Omron CX-Programmer project NewProject (CX-Programmer 9.75)

# PLC NewPLC1: CQM1H CPU51

## Global symbols (name address type ; comment)
0.02 BOOL  ; Up/Down Belts Counter
0.10 BOOL  ; machine reset selector]
0.11 BOOL  ; phc before up/down
0.14 BOOL  ; Enter Movable Roller PHC
100.03 BOOL  ; Open/Close Spendels Box 2
100.05 BOOL  ; Open/Close Spendels Box 1
100.09 BOOL  ; Sarin
100.11 BOOL  ; Green Belts Valve
100.13 BOOL  ; Up/Down Valve
101.00 BOOL  ; arm box 2 run
101.01 BOOL  ; arm box 1 run
101.02 BOOL  ; roller under green belts on box 1
101.03 BOOL  ; Fast Movable Roller Green Belts
101.08 BOOL  ; Roller 1 run
101.10 BOOL  ; UP MACHINE
101.11 BOOL  ; DOWN MACHINE
102.00 BOOL  ; roller2 inverter
102.03 BOOL  ; roller under green belts to box 2
102.05 BOOL  ; Green Belts Down
102.07 BOOL  ; work in box 1
102.09 BOOL  ; Green Belts Run
1.01 BOOL  ; Sensor Arm 2 Opend
1.03 BOOL  ; consent from kiln
1.05 BOOL  ; Sensor Box 2 Exiest
1.06 BOOL  ; Fast Up machine
1.08 BOOL  ; Manual Selector
1.11 BOOL  ; start cycle pb
2.05 BOOL  ; Sensor Arm 1 Opend
2.07 BOOL  ; Sensor Box 1 Exiest
50.07 BOOL  ; Machine Up Slow
50.10 BOOL  ; Machine Down Slow
51.01 BOOL  ; NO START PRESS CYCLE
52.06 BOOL  ; Spendels 2 Rotate run
52.07 BOOL  ; Arm valve (open/close)
52.08 BOOL  ; Green belt run manual
52.09 BOOL  ; Roller 1 run manual
53.04 BOOL  ; Roller 2 run manual
56.01 BOOL  ; machine in floor 60
60.00 BOOL  ; up/down valve on
60.05 BOOL  ; up/down valve manual
60.11 BOOL  ; Green Belts Valve up/down manual
70.11 BOOL  ; Machine Stop in fixed roller
CNT020 BOOL  ; time rotate green belt with roller2 speed
DM416 CHANNEL  ; time rotate green belt with roller2 speed
DM417 CHANNEL  ; time start green belts
DM58 CHANNEL  ; Fixed roller floor
DM59 CHANNEL  ; Machine floor
DM804 CHANNEL  ; box floors count
HR0.00 BOOL  ; Machine automatic
HR0.01 BOOL  ; up/down valve  on
HR0.05 BOOL  ; Machine Down Run
HR1.07 BOOL  ; Green Belts Valve
HR6.00 BOOL  ; box 1 working
HR6.01 BOOL  ; box 2 working
HR93.00 BOOL  ; roller1 run
HR98.03 BOOL  ; box 2 arm valve
HR98.07 BOOL  ; box 1 arm valve
HR99.00 BOOL  ; Machine moving
LR0.11 BOOL  ; Start Cycle hmi
LR1.00 BOOL  ; Spendels  1 rotate
LR1.02 BOOL  ; Green Belts Valve up/down
LR1.03 BOOL  ; Green Belts Rotation
LR1.05 BOOL  ; Slow Up machine
LR1.06 BOOL  ; Fast Up Machine
LR1.10 BOOL  ; Slow Down machine
LR1.11 BOOL  ; Fast  Down machine
LR2.00 BOOL  ; Roller 1 Rotation
LR2.01 BOOL  ; Roller 2 Rotation
LR2.03 BOOL  ; choose box 1
LR2.04 BOOL  ; up/down belts run manual
LR2.05 BOOL  ; Spendels 2 Rotate
LR2.06 BOOL  ; Arm Open
LR2.07 BOOL  ; Arm Close
LR2.08 BOOL  ; choose box 2
LR2.09 BOOL  ; Up/down Valve
TIM006 BOOL  ; time up/down on
TIM016 BOOL  ; machine Stop on fixed roller time
TIM019 BOOL  ; machine stop on fixed roller floor
TIM021 BOOL  ; Arms Not Closed Time
TIM060 BOOL  ; time choose box 1
TIM061 BOOL  ; time choose box 2
TIM299 BOOL  ; Start cycle time

## Program NewProgram1 (no task)

### Section Section1

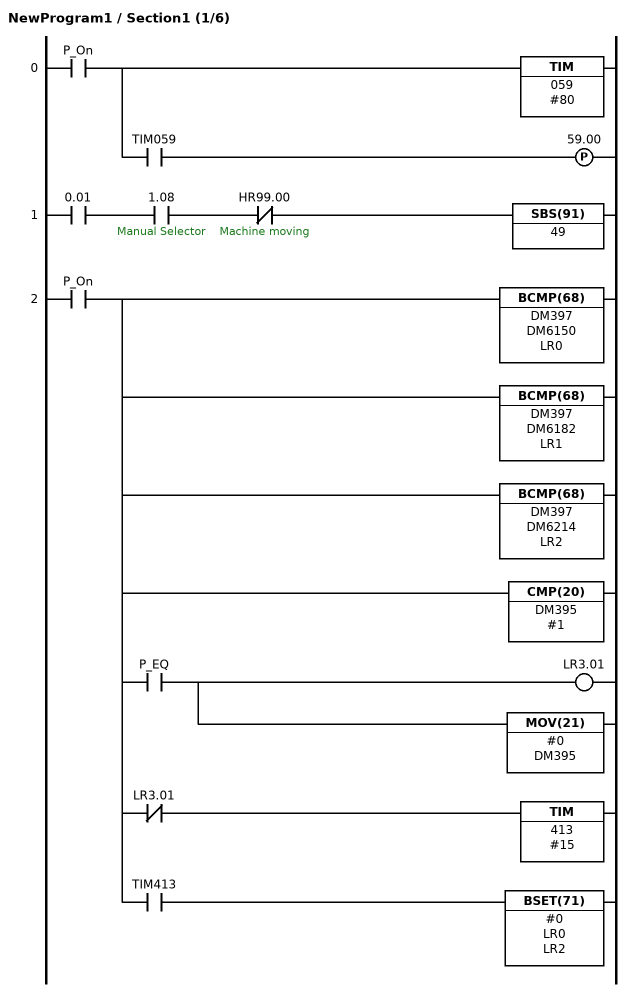
; rung 0
LD P_On
TIM 059 #80
AND TIM059
DIFU(13) 59.00
; rung 1
LD 0.01
AND 1.08  ; Manual Selector
ANDNOT HR99.00  ; Machine moving
SBS(91) 49
; rung 2
LD P_On
OUT TR0
BCMP(68) DM397 DM6150 LR0
BCMP(68) DM397 DM6182 LR1
BCMP(68) DM397 DM6214 LR2
CMP(20) DM395 #1
AND P_EQ
OUT LR3.01
MOV(21) #0 DM395
LD TR0
ANDNOT LR3.01
TIM 413 #15
LD TR0
AND TIM413
BSET(71) #0 LR0 LR2

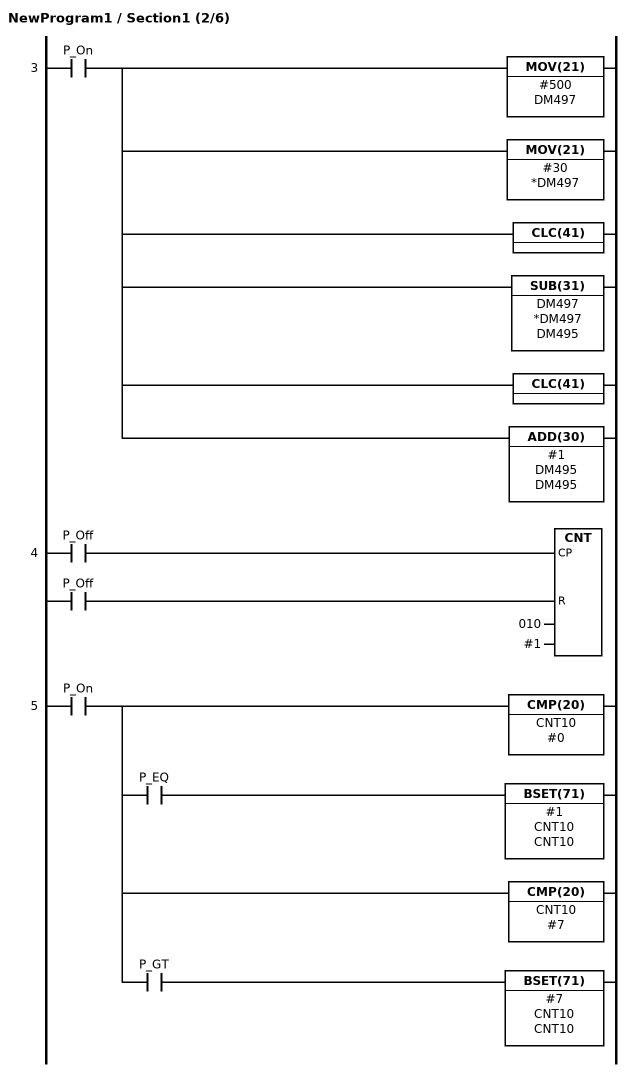
; rung 3
LD P_On
MOV(21) #500 DM497
MOV(21) #30 *DM497
CLC(41)
SUB(31) DM497 *DM497 DM495
CLC(41)
ADD(30) #1 DM495 DM495
; rung 4
LD P_Off
LD P_Off
CNT 010 #1
; rung 5
LD P_On
OUT TR0
CMP(20) CNT10 #0
AND P_EQ
BSET(71) #1 CNT10 CNT10
LD TR0
CMP(20) CNT10 #7
AND P_GT
BSET(71) #7 CNT10 CNT10

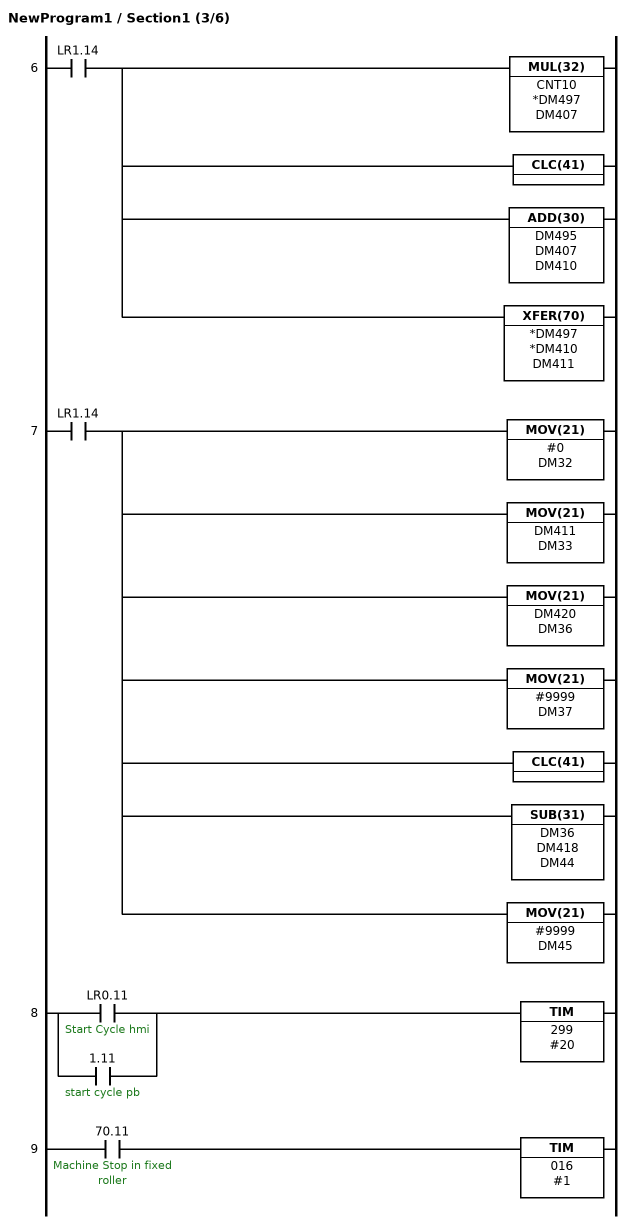
; rung 6
LD LR1.14
MUL(32) CNT10 *DM497 DM407
CLC(41)
ADD(30) DM495 DM407 DM410
XFER(70) *DM497 *DM410 DM411
; rung 7
LD LR1.14
MOV(21) #0 DM32
MOV(21) DM411 DM33
MOV(21) DM420 DM36
MOV(21) #9999 DM37
CLC(41)
SUB(31) DM36 DM418 DM44
MOV(21) #9999 DM45
; rung 8
LD LR0.11  ; Start Cycle hmi
OR 1.11  ; start cycle pb
TIM 299 #20
; rung 9
LD 70.11  ; Machine Stop in fixed roller
TIM 016 #1

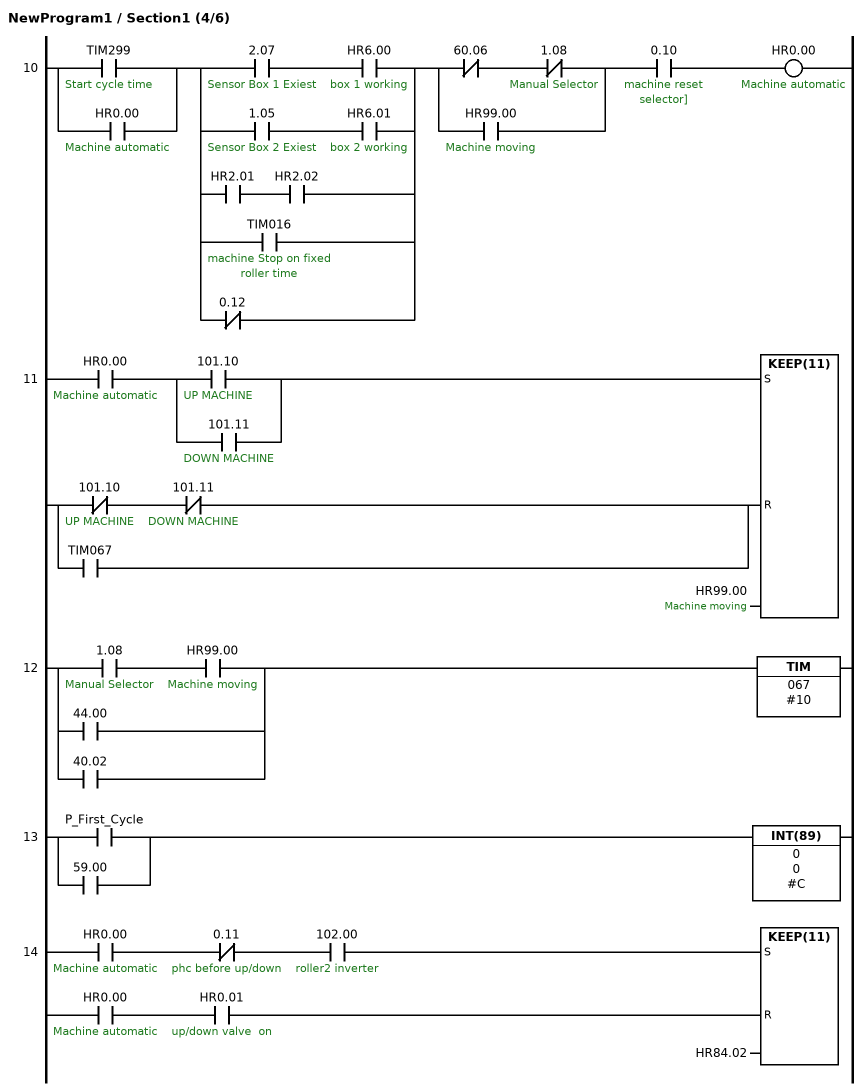
; rung 10
LD TIM299  ; Start cycle time
OR HR0.00  ; Machine automatic
LD 2.07  ; Sensor Box 1 Exiest
AND HR6.00  ; box 1 working
LD 1.05  ; Sensor Box 2 Exiest
AND HR6.01  ; box 2 working
ORLD
LD HR2.01
AND HR2.02
ORLD
OR TIM016  ; machine Stop on fixed roller time
ORNOT 0.12
ANDLD
LDNOT 60.06
ANDNOT 1.08  ; Manual Selector
OR HR99.00  ; Machine moving
ANDLD
AND 0.10  ; machine reset selector]
OUT HR0.00  ; Machine automatic
; rung 11
LD HR0.00  ; Machine automatic
LD 101.10  ; UP MACHINE
OR 101.11  ; DOWN MACHINE
ANDLD
LDNOT 101.10  ; UP MACHINE
ANDNOT 101.11  ; DOWN MACHINE
OR TIM067
KEEP(11) HR99.00  ; Machine moving
; rung 12
LD 1.08  ; Manual Selector
AND HR99.00  ; Machine moving
OR 44.00
OR 40.02
TIM 067 #10
; rung 13
LD P_First_Cycle
OR 59.00
INT(89) 0 0 #C
; rung 14
LD HR0.00  ; Machine automatic
ANDNOT 0.11  ; phc before up/down
AND 102.00  ; roller2 inverter
LD HR0.00  ; Machine automatic
AND HR0.01  ; up/down valve  on
KEEP(11) HR84.02

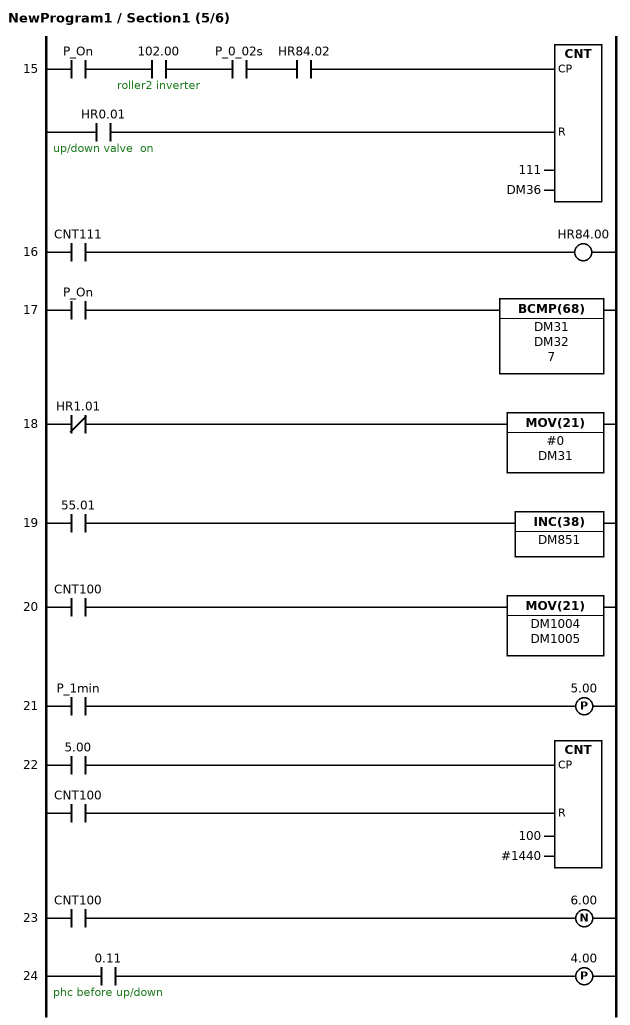
; rung 15
LD P_On
AND 102.00  ; roller2 inverter
AND P_0_02s
AND HR84.02
LD HR0.01  ; up/down valve  on
CNT 111 DM36
; rung 16
LD CNT111
OUT HR84.00
; rung 17
LD P_On
BCMP(68) DM31 DM32 7
; rung 18
LDNOT HR1.01
MOV(21) #0 DM31
; rung 19
LD 55.01
INC(38) DM851
; rung 20
LD CNT100
MOV(21) DM1004 DM1005
; rung 21
LD P_1min
DIFU(13) 5.00
; rung 22
LD 5.00
LD CNT100
CNT 100 #1440
; rung 23
LD CNT100
DIFD(14) 6.00
; rung 24
LD 0.11  ; phc before up/down
DIFU(13) 4.00

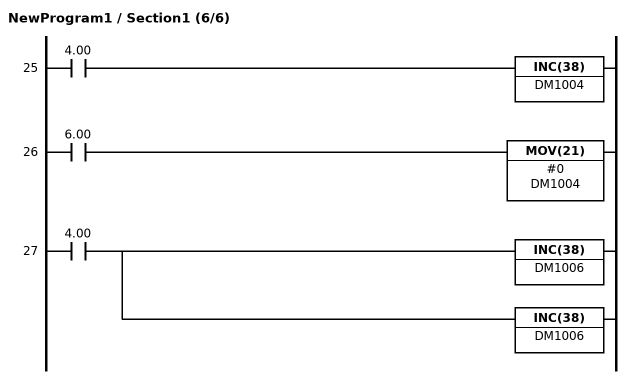
; rung 25
LD 4.00
INC(38) DM1004
; rung 26
LD 6.00
MOV(21) #0 DM1004
; rung 27
LD 4.00
INC(38) DM1006
INC(38) DM1006

### Section Section2

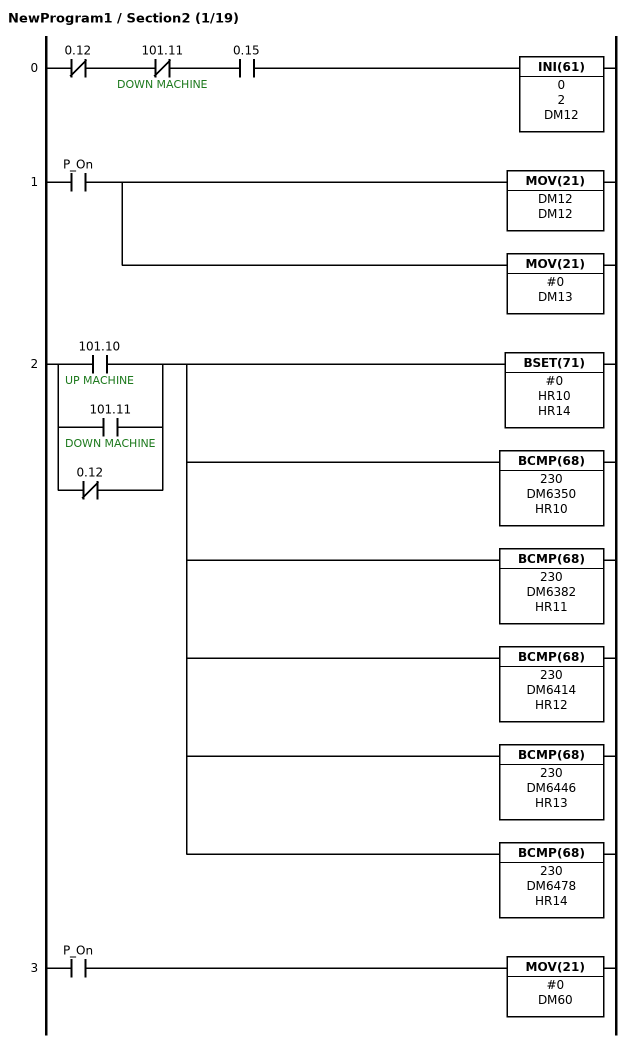
; rung 0
LDNOT 0.12
ANDNOT 101.11  ; DOWN MACHINE
AND 0.15
INI(61) 0 2 DM12
; rung 1
LD P_On
MOV(21) DM12 DM12
MOV(21) #0 DM13
; rung 2
LD 101.10  ; UP MACHINE
OR 101.11  ; DOWN MACHINE
ORNOT 0.12
BSET(71) #0 HR10 HR14
BCMP(68) 230 DM6350 HR10
BCMP(68) 230 DM6382 HR11
BCMP(68) 230 DM6414 HR12
BCMP(68) 230 DM6446 HR13
BCMP(68) 230 DM6478 HR14
; rung 3
LD P_On
MOV(21) #0 DM60

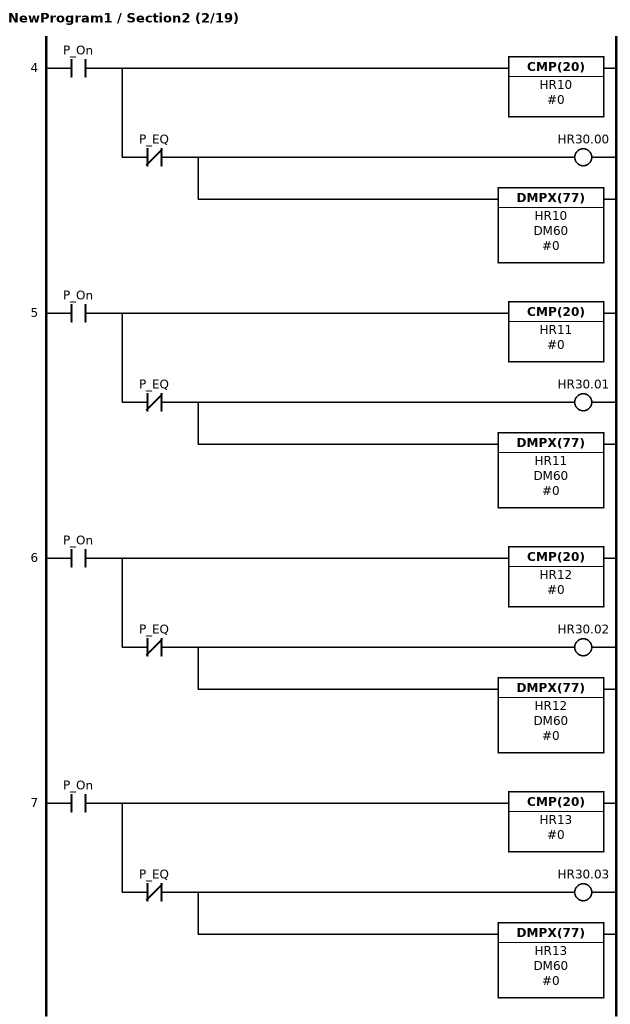
; rung 4
LD P_On
CMP(20) HR10 #0
ANDNOT P_EQ
OUT HR30.00
DMPX(77) HR10 DM60 #0
; rung 5
LD P_On
CMP(20) HR11 #0
ANDNOT P_EQ
OUT HR30.01
DMPX(77) HR11 DM60 #0
; rung 6
LD P_On
CMP(20) HR12 #0
ANDNOT P_EQ
OUT HR30.02
DMPX(77) HR12 DM60 #0
; rung 7
LD P_On
CMP(20) HR13 #0
ANDNOT P_EQ
OUT HR30.03
DMPX(77) HR13 DM60 #0

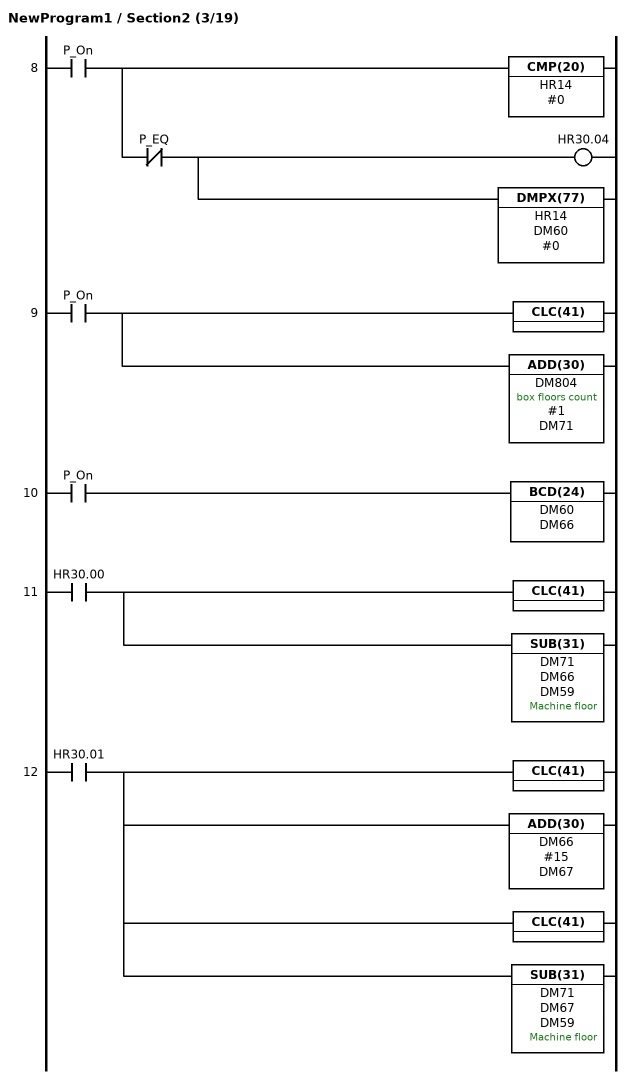
; rung 8
LD P_On
CMP(20) HR14 #0
ANDNOT P_EQ
OUT HR30.04
DMPX(77) HR14 DM60 #0
; rung 9
LD P_On
CLC(41)
ADD(30) DM804 #1 DM71  ; box floors count
; rung 10
LD P_On
BCD(24) DM60 DM66
; rung 11
LD HR30.00
CLC(41)
SUB(31) DM71 DM66 DM59  ; Machine floor
; rung 12
LD HR30.01
CLC(41)
ADD(30) DM66 #15 DM67
CLC(41)
SUB(31) DM71 DM67 DM59  ; Machine floor

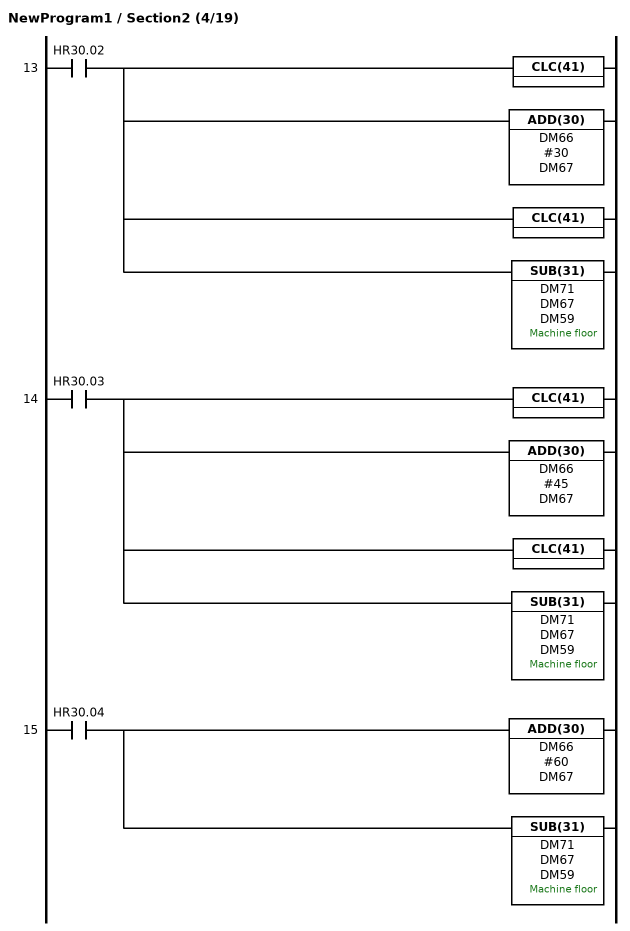
; rung 13
LD HR30.02
CLC(41)
ADD(30) DM66 #30 DM67
CLC(41)
SUB(31) DM71 DM67 DM59  ; Machine floor
; rung 14
LD HR30.03
CLC(41)
ADD(30) DM66 #45 DM67
CLC(41)
SUB(31) DM71 DM67 DM59  ; Machine floor
; rung 15
LD HR30.04
ADD(30) DM66 #60 DM67
SUB(31) DM71 DM67 DM59  ; Machine floor

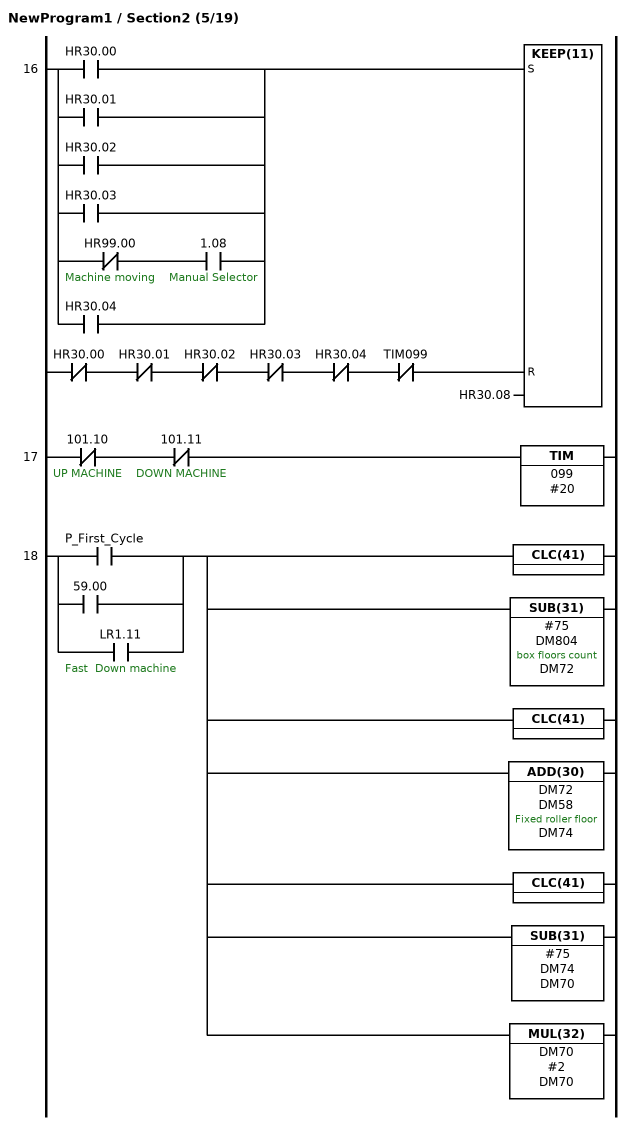
; rung 16
LD HR30.00
OR HR30.01
OR HR30.02
OR HR30.03
LDNOT HR99.00  ; Machine moving
AND 1.08  ; Manual Selector
ORLD
OR HR30.04
LDNOT HR30.00
ANDNOT HR30.01
ANDNOT HR30.02
ANDNOT HR30.03
ANDNOT HR30.04
ANDNOT TIM099
KEEP(11) HR30.08
; rung 17
LDNOT 101.10  ; UP MACHINE
ANDNOT 101.11  ; DOWN MACHINE
TIM 099 #20
; rung 18
LD P_First_Cycle
OR 59.00
OR LR1.11  ; Fast  Down machine
CLC(41)
SUB(31) #75 DM804 DM72  ; box floors count
CLC(41)
ADD(30) DM72 DM58 DM74  ; Fixed roller floor
CLC(41)
SUB(31) #75 DM74 DM70
MUL(32) DM70 #2 DM70

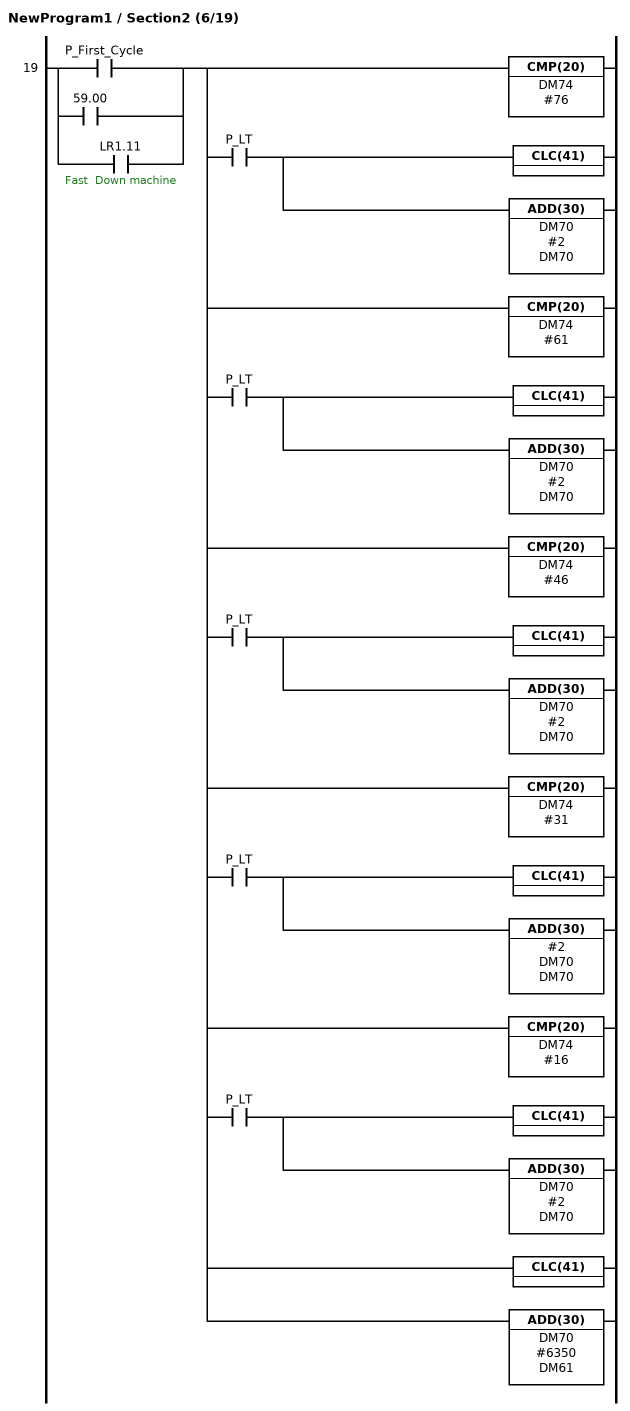
; rung 19
LD P_First_Cycle
OR 59.00
OR LR1.11  ; Fast  Down machine
OUT TR0
CMP(20) DM74 #76
AND P_LT
CLC(41)
ADD(30) DM70 #2 DM70
LD TR0
CMP(20) DM74 #61
AND P_LT
CLC(41)
ADD(30) DM70 #2 DM70
LD TR0
CMP(20) DM74 #46
AND P_LT
CLC(41)
ADD(30) DM70 #2 DM70
LD TR0
CMP(20) DM74 #31
AND P_LT
CLC(41)
ADD(30) #2 DM70 DM70
LD TR0
CMP(20) DM74 #16
AND P_LT
CLC(41)
ADD(30) DM70 #2 DM70
LD TR0
CLC(41)
ADD(30) DM70 #6350 DM61

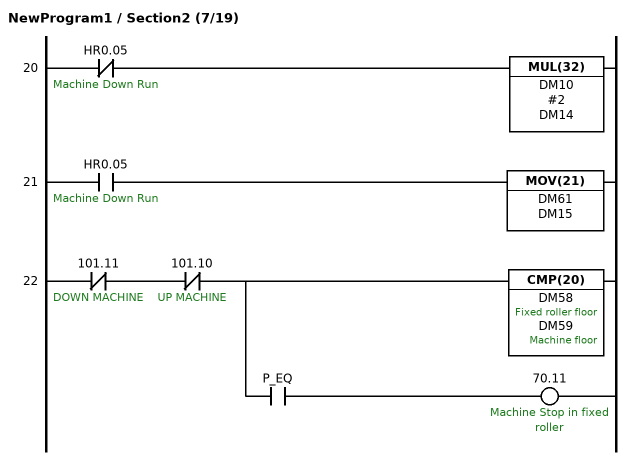
; rung 20
LDNOT HR0.05  ; Machine Down Run
MUL(32) DM10 #2 DM14
; rung 21
LD HR0.05  ; Machine Down Run
MOV(21) DM61 DM15
; rung 22
LDNOT 101.11  ; DOWN MACHINE
ANDNOT 101.10  ; UP MACHINE
CMP(20) DM58 DM59  ; Fixed roller floor, Machine floor
AND P_EQ
OUT 70.11  ; Machine Stop in fixed roller

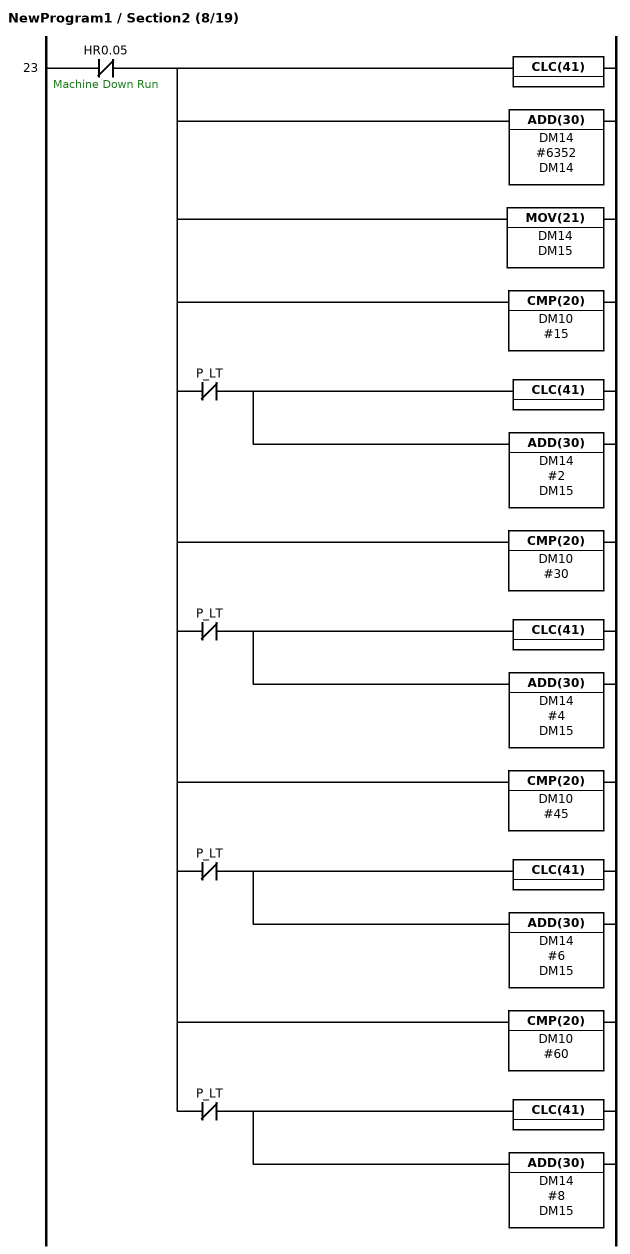
; rung 23
LDNOT HR0.05  ; Machine Down Run
OUT TR0
CLC(41)
ADD(30) DM14 #6352 DM14
MOV(21) DM14 DM15
CMP(20) DM10 #15
ANDNOT P_LT
CLC(41)
ADD(30) DM14 #2 DM15
LD TR0
CMP(20) DM10 #30
ANDNOT P_LT
CLC(41)
ADD(30) DM14 #4 DM15
LD TR0
CMP(20) DM10 #45
ANDNOT P_LT
CLC(41)
ADD(30) DM14 #6 DM15
LD TR0
CMP(20) DM10 #60
ANDNOT P_LT
CLC(41)
ADD(30) DM14 #8 DM15

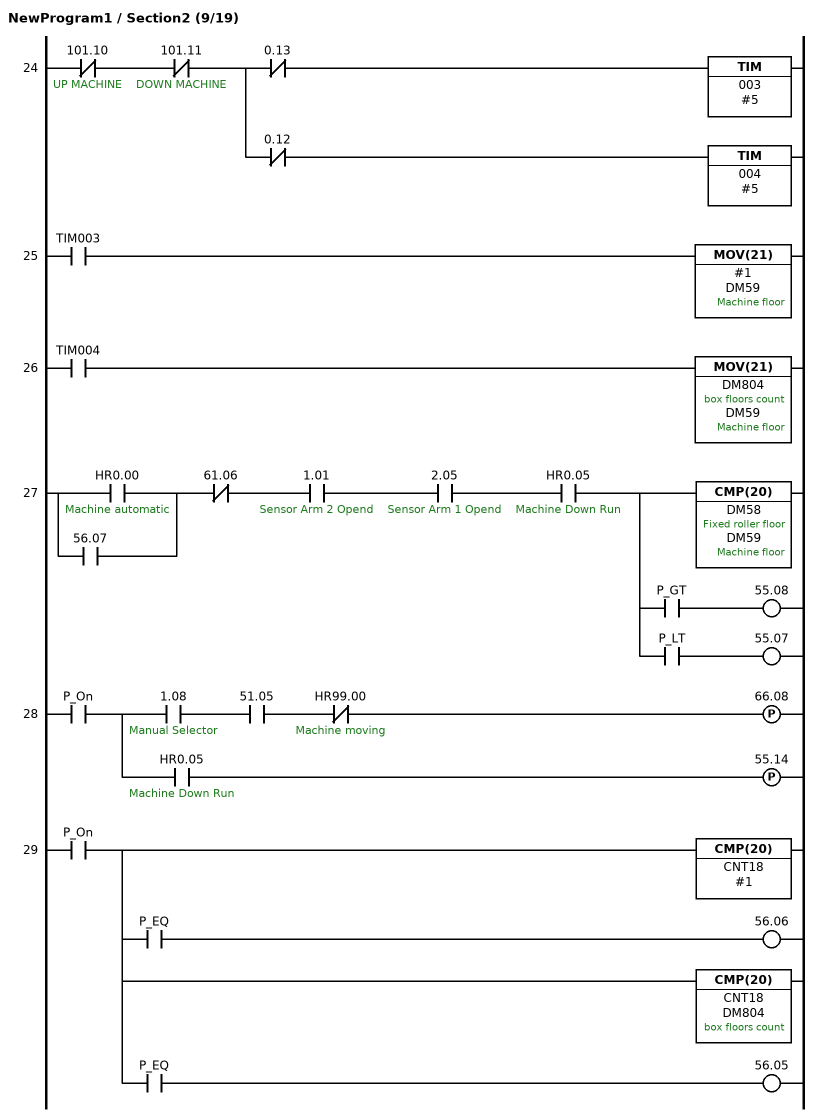
; rung 24
LDNOT 101.10  ; UP MACHINE
ANDNOT 101.11  ; DOWN MACHINE
OUT TR0
ANDNOT 0.13
TIM 003 #5
LD TR0
ANDNOT 0.12
TIM 004 #5
; rung 25
LD TIM003
MOV(21) #1 DM59  ; Machine floor
; rung 26
LD TIM004
MOV(21) DM804 DM59  ; box floors count, Machine floor
; rung 27
LD HR0.00  ; Machine automatic
OR 56.07
ANDNOT 61.06
AND 1.01  ; Sensor Arm 2 Opend
AND 2.05  ; Sensor Arm 1 Opend
AND HR0.05  ; Machine Down Run
OUT TR0
CMP(20) DM58 DM59  ; Fixed roller floor, Machine floor
AND P_GT
OUT 55.08
LD TR0
AND P_LT
OUT 55.07
; rung 28
LD P_On
OUT TR0
AND 1.08  ; Manual Selector
AND 51.05
ANDNOT HR99.00  ; Machine moving
DIFU(13) 66.08
LD TR0
AND HR0.05  ; Machine Down Run
DIFU(13) 55.14
; rung 29
LD P_On
OUT TR0
CMP(20) CNT18 #1
AND P_EQ
OUT 56.06
LD TR0
CMP(20) CNT18 DM804  ; box floors count
AND P_EQ
OUT 56.05

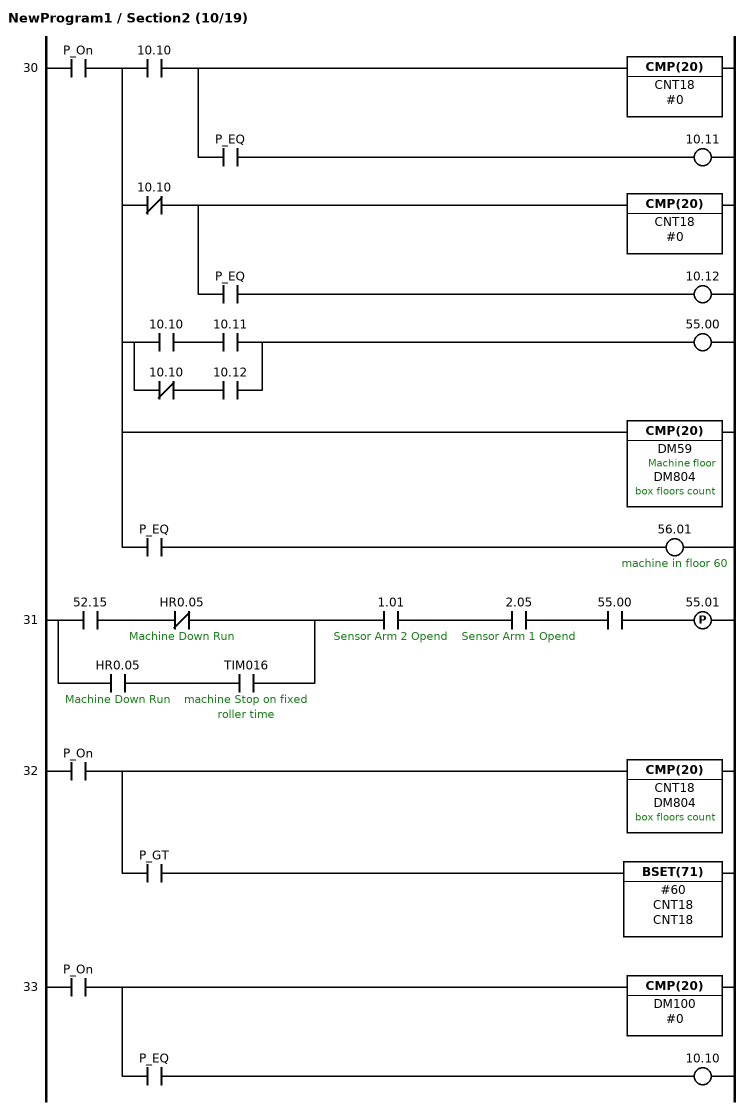
; rung 30
LD P_On
OUT TR0
AND 10.10
CMP(20) CNT18 #0
AND P_EQ
OUT 10.11
LD TR0
ANDNOT 10.10
CMP(20) CNT18 #0
AND P_EQ
OUT 10.12
LD TR0
LD 10.10
AND 10.11
LDNOT 10.10
AND 10.12
ORLD
ANDLD
OUT 55.00
LD TR0
CMP(20) DM59 DM804  ; Machine floor, box floors count
AND P_EQ
OUT 56.01  ; machine in floor 60
; rung 31
LD 52.15
ANDNOT HR0.05  ; Machine Down Run
LD HR0.05  ; Machine Down Run
AND TIM016  ; machine Stop on fixed roller time
ORLD
AND 1.01  ; Sensor Arm 2 Opend
AND 2.05  ; Sensor Arm 1 Opend
AND 55.00
DIFU(13) 55.01
; rung 32
LD P_On
CMP(20) CNT18 DM804  ; box floors count
AND P_GT
BSET(71) #60 CNT18 CNT18
; rung 33
LD P_On
CMP(20) DM100 #0
AND P_EQ
OUT 10.10

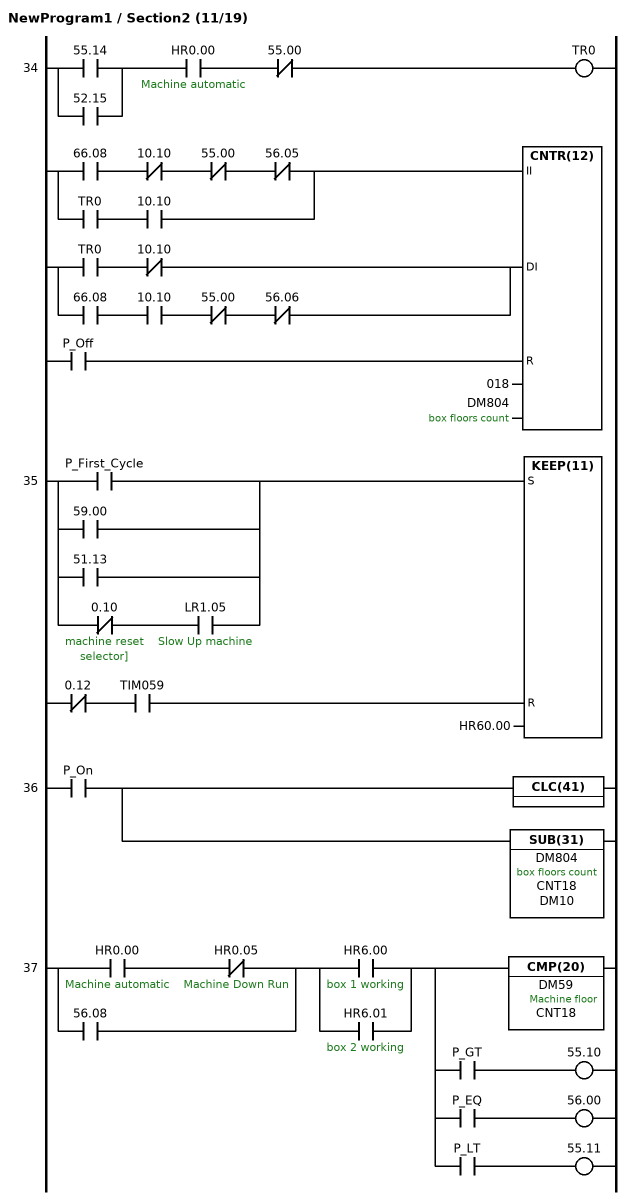
; rung 34
LD 66.08
ANDNOT 10.10
ANDNOT 55.00
ANDNOT 56.05
LD 55.14
OR 52.15
AND HR0.00  ; Machine automatic
ANDNOT 55.00
OUT TR0
AND 10.10
ORLD
LD TR0
ANDNOT 10.10
LD 66.08
AND 10.10
ANDNOT 55.00
ANDNOT 56.06
ORLD
LD P_Off
CNTR(12) 018 DM804  ; box floors count
; rung 35
LD P_First_Cycle
OR 59.00
OR 51.13
LDNOT 0.10  ; machine reset selector]
AND LR1.05  ; Slow Up machine
ORLD
LDNOT 0.12
AND TIM059
KEEP(11) HR60.00
; rung 36
LD P_On
CLC(41)
SUB(31) DM804 CNT18 DM10  ; box floors count
; rung 37
LD HR0.00  ; Machine automatic
ANDNOT HR0.05  ; Machine Down Run
OR 56.08
LD HR6.00  ; box 1 working
OR HR6.01  ; box 2 working
ANDLD
OUT TR0
CMP(20) DM59 CNT18  ; Machine floor
AND P_GT
OUT 55.10
LD TR0
AND P_EQ
OUT 56.00
LD TR0
AND P_LT
OUT 55.11

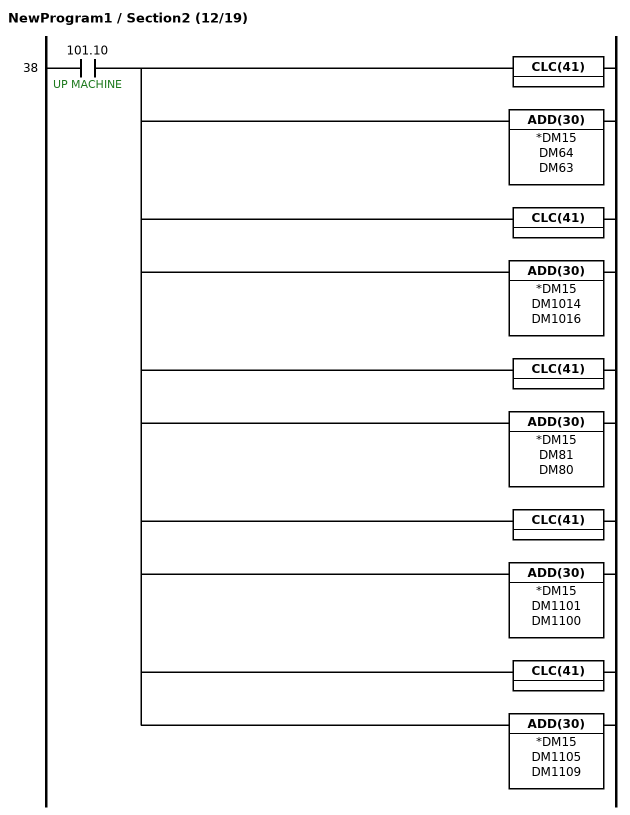
; rung 38
LD 101.10  ; UP MACHINE
CLC(41)
ADD(30) *DM15 DM64 DM63
CLC(41)
ADD(30) *DM15 DM1014 DM1016
CLC(41)
ADD(30) *DM15 DM81 DM80
CLC(41)
ADD(30) *DM15 DM1101 DM1100
CLC(41)
ADD(30) *DM15 DM1105 DM1109

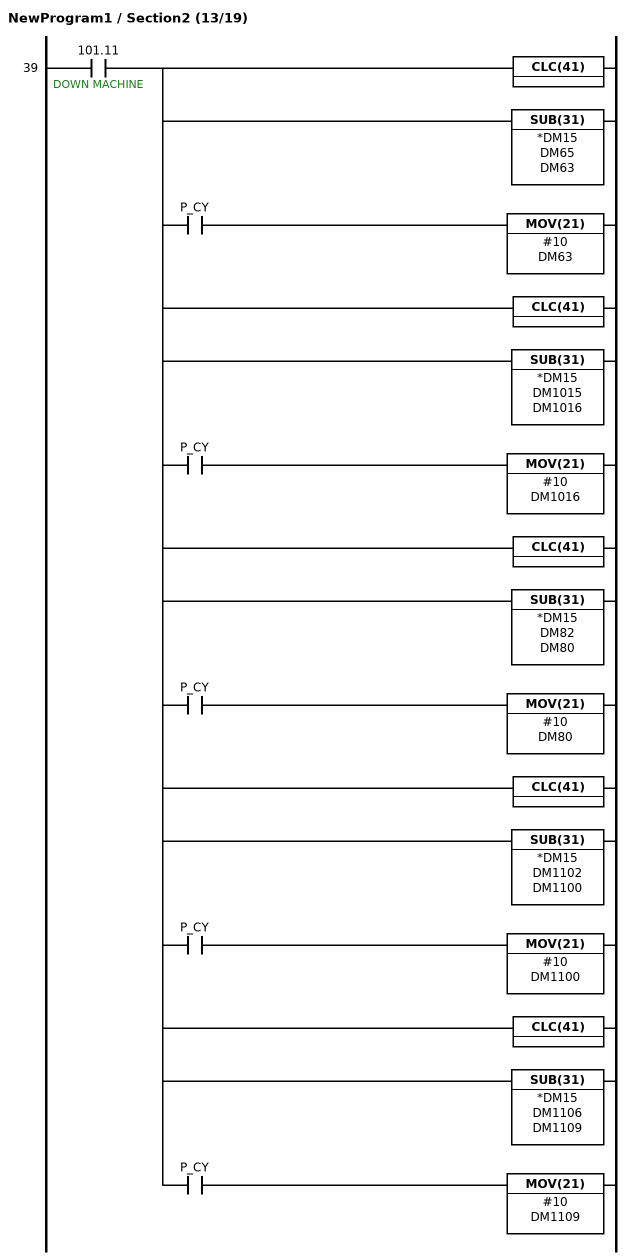
; rung 39
LD 101.11  ; DOWN MACHINE
OUT TR0
CLC(41)
SUB(31) *DM15 DM65 DM63
AND P_CY
MOV(21) #10 DM63
LD TR0
CLC(41)
SUB(31) *DM15 DM1015 DM1016
AND P_CY
MOV(21) #10 DM1016
LD TR0
CLC(41)
SUB(31) *DM15 DM82 DM80
AND P_CY
MOV(21) #10 DM80
LD TR0
CLC(41)
SUB(31) *DM15 DM1102 DM1100
AND P_CY
MOV(21) #10 DM1100
LD TR0
CLC(41)
SUB(31) *DM15 DM1106 DM1109
AND P_CY
MOV(21) #10 DM1109

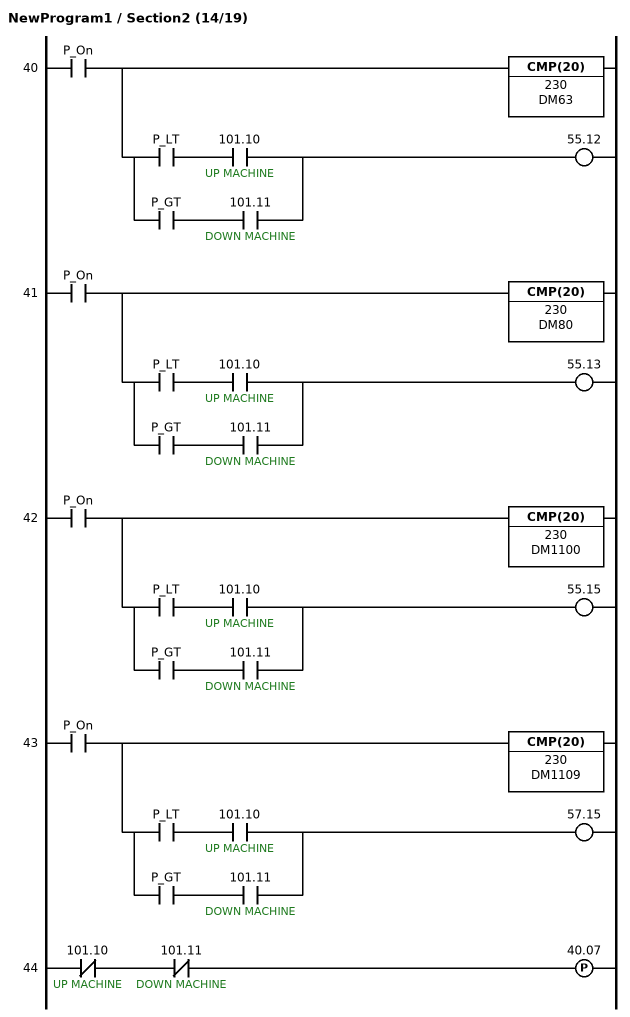
; rung 40
LD P_On
CMP(20) 230 DM63
LD P_LT
AND 101.10  ; UP MACHINE
LD P_GT
AND 101.11  ; DOWN MACHINE
ORLD
ANDLD
OUT 55.12
; rung 41
LD P_On
CMP(20) 230 DM80
LD P_LT
AND 101.10  ; UP MACHINE
LD P_GT
AND 101.11  ; DOWN MACHINE
ORLD
ANDLD
OUT 55.13
; rung 42
LD P_On
CMP(20) 230 DM1100
LD P_LT
AND 101.10  ; UP MACHINE
LD P_GT
AND 101.11  ; DOWN MACHINE
ORLD
ANDLD
OUT 55.15
; rung 43
LD P_On
CMP(20) 230 DM1109
LD P_LT
AND 101.10  ; UP MACHINE
LD P_GT
AND 101.11  ; DOWN MACHINE
ORLD
ANDLD
OUT 57.15
; rung 44
LDNOT 101.10  ; UP MACHINE
ANDNOT 101.11  ; DOWN MACHINE
DIFU(13) 40.07

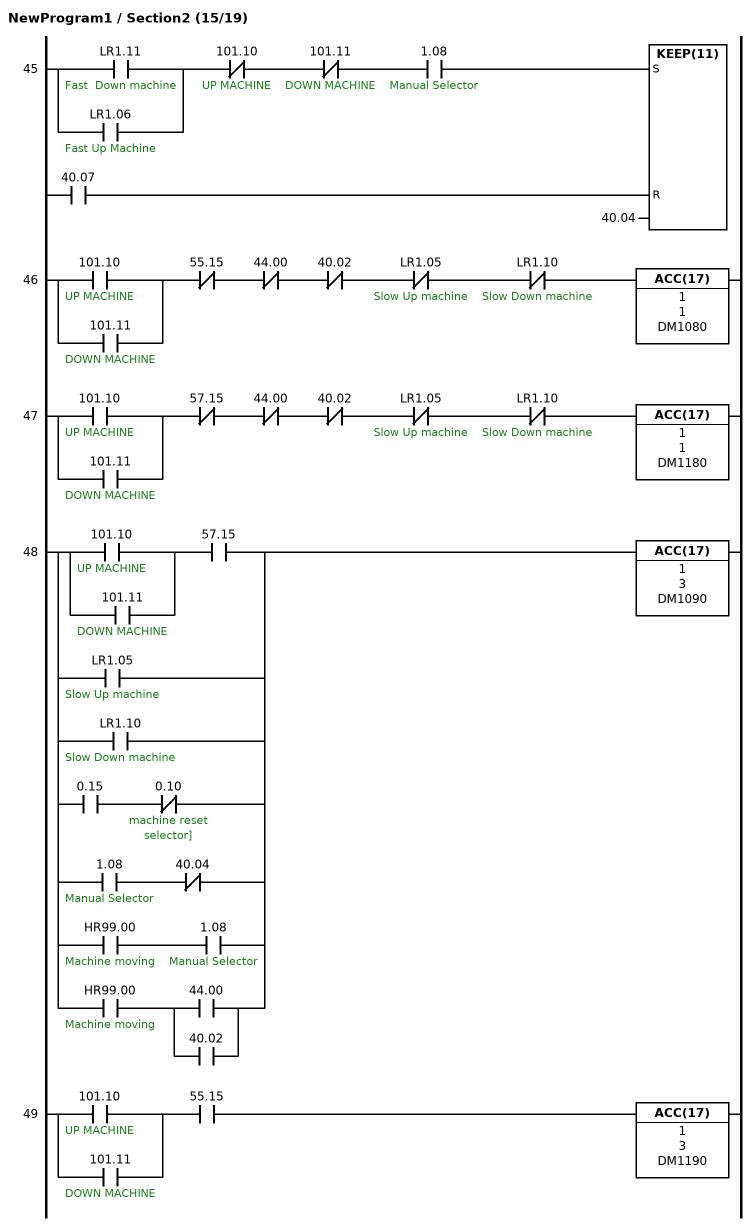
; rung 45
LD LR1.11  ; Fast  Down machine
OR LR1.06  ; Fast Up Machine
ANDNOT 101.10  ; UP MACHINE
ANDNOT 101.11  ; DOWN MACHINE
AND 1.08  ; Manual Selector
LD 40.07
KEEP(11) 40.04
; rung 46
LD 101.10  ; UP MACHINE
OR 101.11  ; DOWN MACHINE
ANDNOT 55.15
ANDNOT 44.00
ANDNOT 40.02
ANDNOT LR1.05  ; Slow Up machine
ANDNOT LR1.10  ; Slow Down machine
ACC(17) 1 1 DM1080
; rung 47
LD 101.10  ; UP MACHINE
OR 101.11  ; DOWN MACHINE
ANDNOT 57.15
ANDNOT 44.00
ANDNOT 40.02
ANDNOT LR1.05  ; Slow Up machine
ANDNOT LR1.10  ; Slow Down machine
ACC(17) 1 1 DM1180
; rung 48
LD 101.10  ; UP MACHINE
OR 101.11  ; DOWN MACHINE
AND 57.15
OR LR1.05  ; Slow Up machine
OR LR1.10  ; Slow Down machine
LD 0.15
ANDNOT 0.10  ; machine reset selector]
ORLD
LD 1.08  ; Manual Selector
ANDNOT 40.04
ORLD
LD HR99.00  ; Machine moving
AND 1.08  ; Manual Selector
ORLD
LD HR99.00  ; Machine moving
LD 44.00
OR 40.02
ANDLD
ORLD
ACC(17) 1 3 DM1090
; rung 49
LD 101.10  ; UP MACHINE
OR 101.11  ; DOWN MACHINE
AND 55.15
ACC(17) 1 3 DM1190

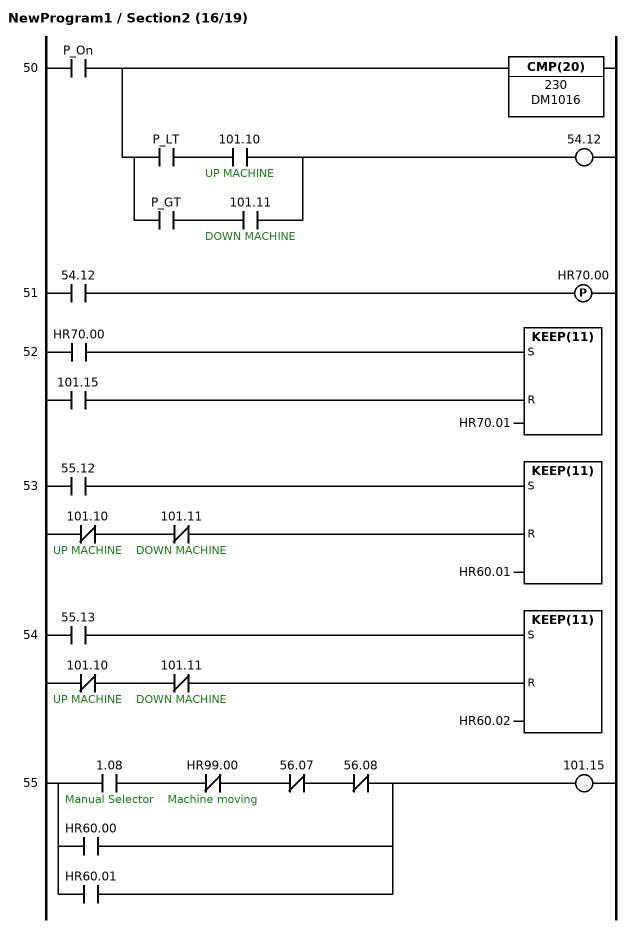
; rung 50
LD P_On
CMP(20) 230 DM1016
LD P_LT
AND 101.10  ; UP MACHINE
LD P_GT
AND 101.11  ; DOWN MACHINE
ORLD
ANDLD
OUT 54.12
; rung 51
LD 54.12
DIFU(13) HR70.00
; rung 52
LD HR70.00
LD 101.15
KEEP(11) HR70.01
; rung 53
LD 55.12
LDNOT 101.10  ; UP MACHINE
ANDNOT 101.11  ; DOWN MACHINE
KEEP(11) HR60.01
; rung 54
LD 55.13
LDNOT 101.10  ; UP MACHINE
ANDNOT 101.11  ; DOWN MACHINE
KEEP(11) HR60.02
; rung 55
LD 1.08  ; Manual Selector
ANDNOT HR99.00  ; Machine moving
ANDNOT 56.07
ANDNOT 56.08
OR HR60.00
OR HR60.01
OUT 101.15

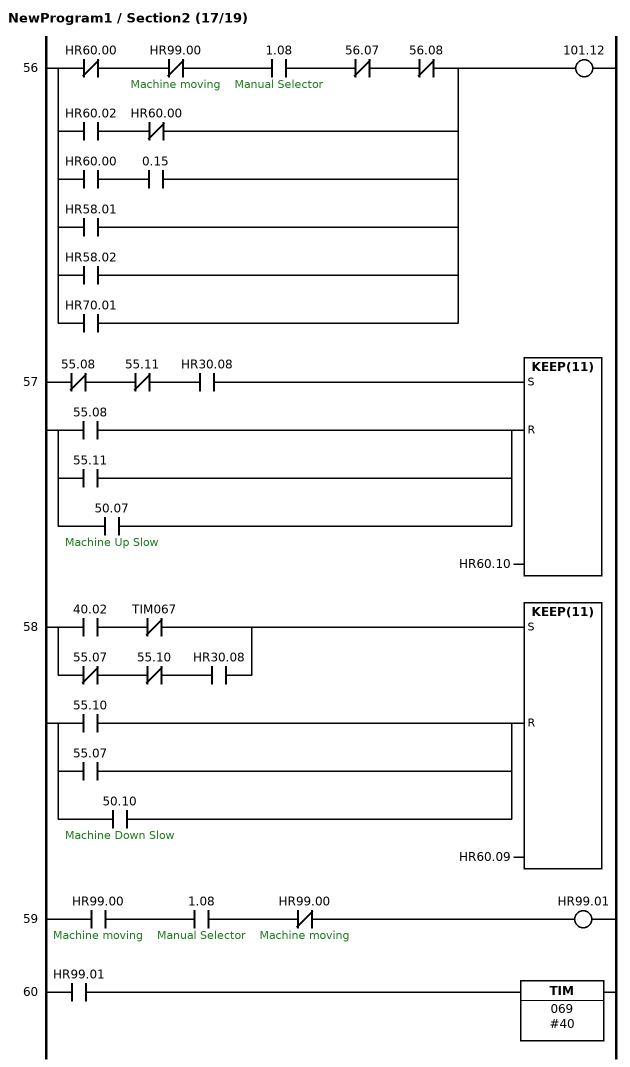
; rung 56
LDNOT HR60.00
ANDNOT HR99.00  ; Machine moving
AND 1.08  ; Manual Selector
ANDNOT 56.07
ANDNOT 56.08
LD HR60.02
ANDNOT HR60.00
ORLD
LD HR60.00
AND 0.15
ORLD
OR HR58.01
OR HR58.02
OR HR70.01
OUT 101.12
; rung 57
LDNOT 55.08
ANDNOT 55.11
AND HR30.08
LD 55.08
OR 55.11
OR 50.07  ; Machine Up Slow
KEEP(11) HR60.10
; rung 58
LD 40.02
ANDNOT TIM067
LDNOT 55.07
ANDNOT 55.10
AND HR30.08
ORLD
LD 55.10
OR 55.07
OR 50.10  ; Machine Down Slow
KEEP(11) HR60.09
; rung 59
LD HR99.00  ; Machine moving
AND 1.08  ; Manual Selector
ANDNOT HR99.00  ; Machine moving
OUT HR99.01
; rung 60
LD HR99.01
TIM 069 #40

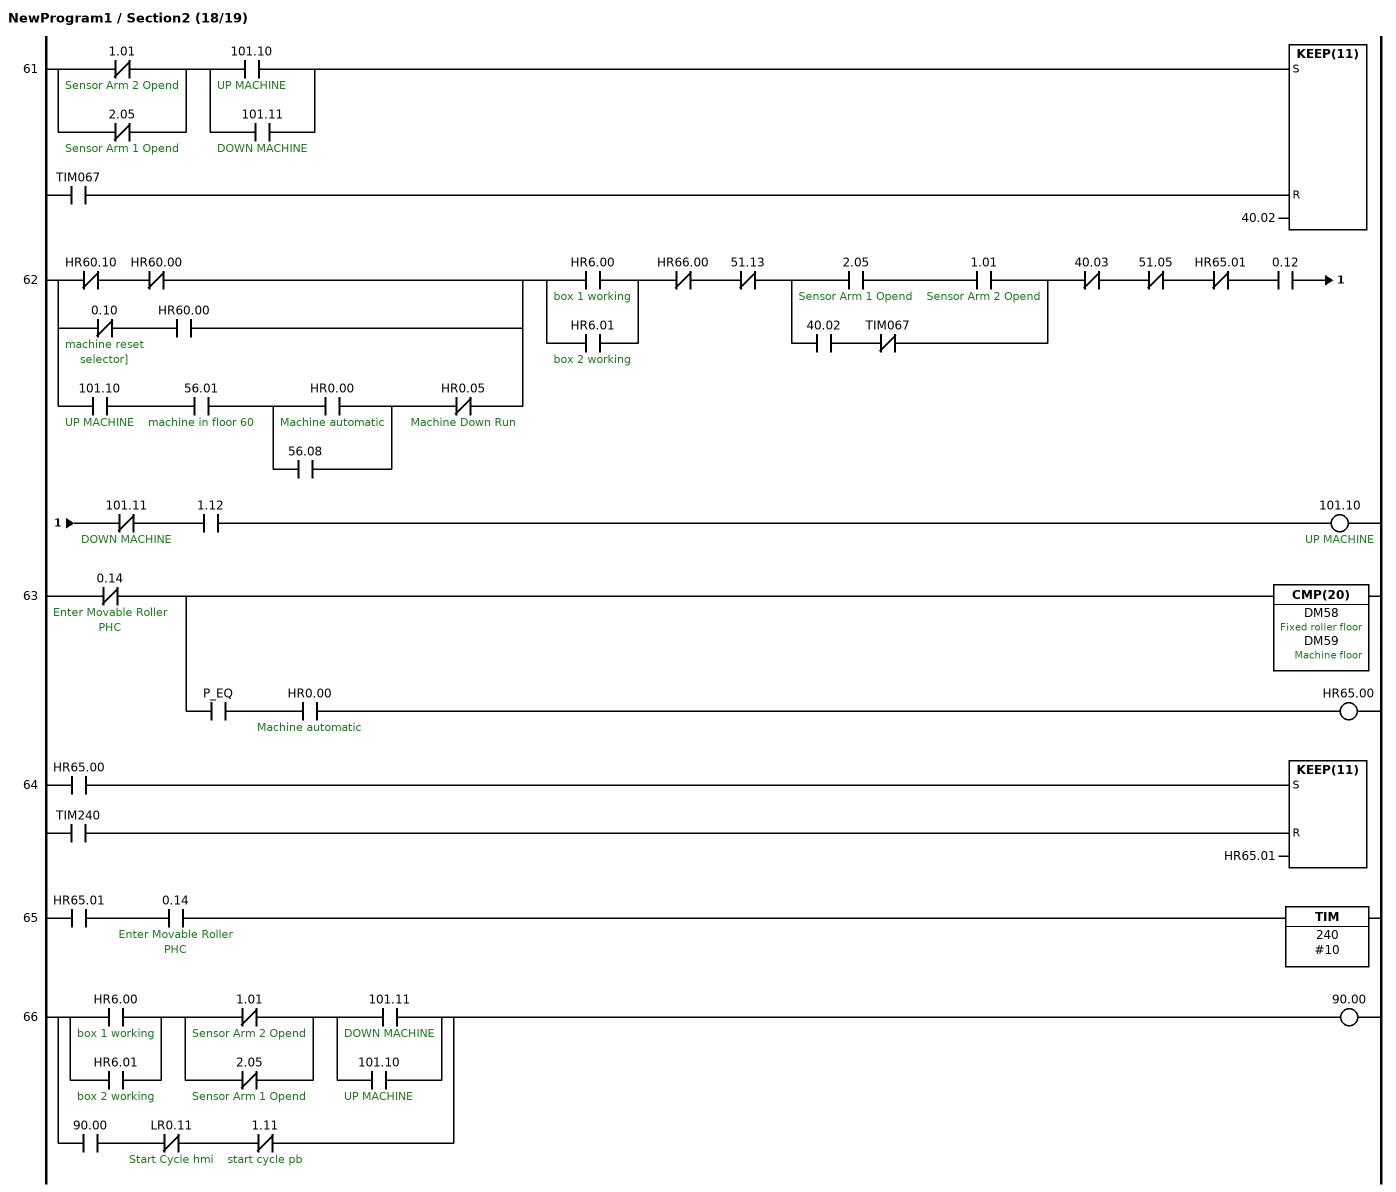
; rung 61
LDNOT 1.01  ; Sensor Arm 2 Opend
ORNOT 2.05  ; Sensor Arm 1 Opend
LD 101.10  ; UP MACHINE
OR 101.11  ; DOWN MACHINE
ANDLD
LD TIM067
KEEP(11) 40.02
; rung 62
LDNOT HR60.10
ANDNOT HR60.00
LDNOT 0.10  ; machine reset selector]
AND HR60.00
ORLD
LD 101.10  ; UP MACHINE
AND 56.01  ; machine in floor 60
LD HR0.00  ; Machine automatic
OR 56.08
ANDLD
ANDNOT HR0.05  ; Machine Down Run
ORLD
LD HR6.00  ; box 1 working
OR HR6.01  ; box 2 working
ANDLD
ANDNOT HR66.00
ANDNOT 51.13
LD 2.05  ; Sensor Arm 1 Opend
AND 1.01  ; Sensor Arm 2 Opend
LD 40.02
ANDNOT TIM067
ORLD
ANDLD
ANDNOT 40.03
ANDNOT 51.05
ANDNOT HR65.01
AND 0.12
ANDNOT 101.11  ; DOWN MACHINE
AND 1.12
OUT 101.10  ; UP MACHINE
; rung 63
LDNOT 0.14  ; Enter Movable Roller PHC
CMP(20) DM58 DM59  ; Fixed roller floor, Machine floor
AND P_EQ
AND HR0.00  ; Machine automatic
OUT HR65.00
; rung 64
LD HR65.00
LD TIM240
KEEP(11) HR65.01
; rung 65
LD HR65.01
AND 0.14  ; Enter Movable Roller PHC
TIM 240 #10
; rung 66
LD HR6.00  ; box 1 working
OR HR6.01  ; box 2 working
LDNOT 1.01  ; Sensor Arm 2 Opend
ORNOT 2.05  ; Sensor Arm 1 Opend
ANDLD
LD 101.11  ; DOWN MACHINE
OR 101.10  ; UP MACHINE
ANDLD
LD 90.00
ANDNOT LR0.11  ; Start Cycle hmi
ANDNOT 1.11  ; start cycle pb
ORLD
OUT 90.00

